Omron CX-Programmer project 新工程 (CX-Programmer 9.42)

# PLC 新PLC1: CP1H XA

## Global symbols (name address type ; comment)
0.00 BOOL  ; 启动按钮
0.01 BOOL  ; 停止按钮
10.00 BOOL  ; 东西绿灯20s+闪3s
10.01 BOOL  ; 东西黄灯2s
10.02 BOOL  ; 东西红灯25s
10.03 BOOL  ; 南北绿灯20s+闪3s
10.04 BOOL  ; 南北黄灯2s
10.05 BOOL  ; 南北红灯25s

## Program 新程序1 (cyclic task 0)

### Section 段1

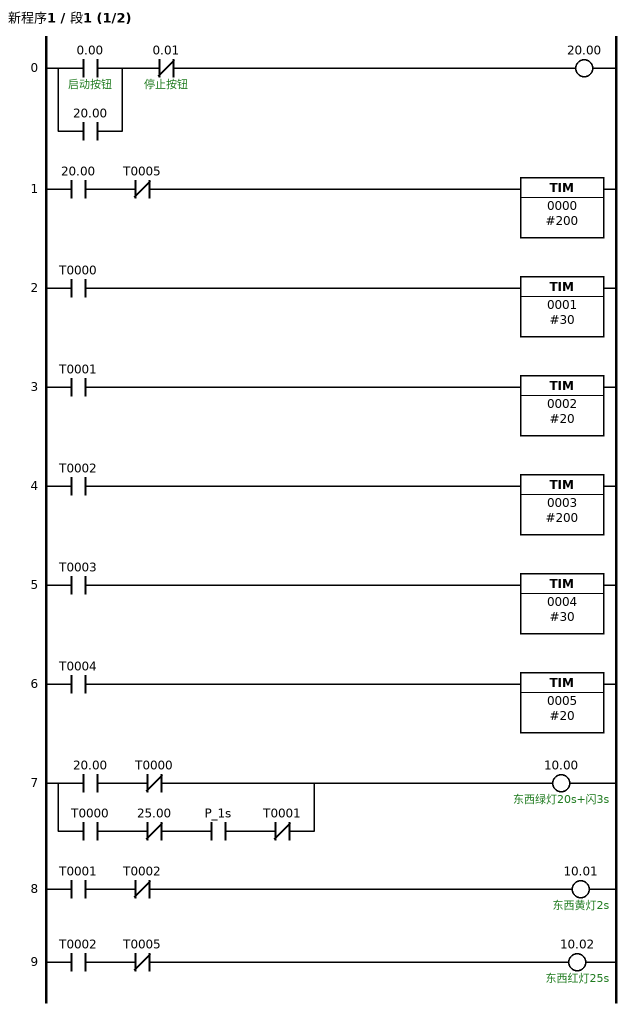
; rung 0
LD 0.00  ; 启动按钮
OR 20.00
ANDNOT 0.01  ; 停止按钮
OUT 20.00
; rung 1
LD 20.00
ANDNOT T0005
TIM 0000 #200
; rung 2
LD T0000
TIM 0001 #30
; rung 3
LD T0001
TIM 0002 #20
; rung 4
LD T0002
TIM 0003 #200
; rung 5
LD T0003
TIM 0004 #30
; rung 6
LD T0004
TIM 0005 #20
; rung 7
LD 20.00
ANDNOT T0000
LD T0000
ANDNOT 25.00
AND P_1s
ANDNOT T0001
ORLD
OUT 10.00  ; 东西绿灯20s+闪3s
; rung 8
LD T0001
ANDNOT T0002
OUT 10.01  ; 东西黄灯2s
; rung 9
LD T0002
ANDNOT T0005
OUT 10.02  ; 东西红灯25s

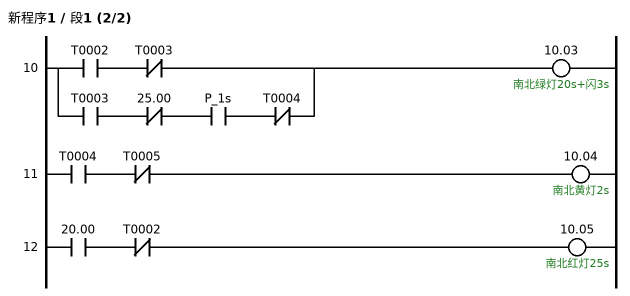
; rung 10
LD T0002
ANDNOT T0003
LD T0003
ANDNOT 25.00
AND P_1s
ANDNOT T0004
ORLD
OUT 10.03  ; 南北绿灯20s+闪3s
; rung 11
LD T0004
ANDNOT T0005
OUT 10.04  ; 南北黄灯2s
; rung 12
LD 20.00
ANDNOT T0002
OUT 10.05  ; 南北红灯25s

### Section END
; rung 0
END(001)